PROGRAM DataTypes
VAR
	floatExample : REAL;
	someStr : STRING;
	someInt : INT := 20;
	{REFERENCE TO someInt}
	refInt : REFERENCE TO INT REF=someInt;
	
	bytesCountFloat : UINT;
	bytesCountInt : UINT;
	bytesCountStr : UINT;
	
	{U may declare negative indexes : [-5..4]}
	someArr : ARRAY[1..5] OF INT := [10, 20, 30, 40, 50];
	twoDemArr : ARRAY [0..3, 0..9] OF REAL;
END_VAR

bytesCountFloat := SIZEOF(floatExample);
bytesCountStr := SIZEOF(someStr);
bytesCountInt := SIZEOF(someInt);

someArr[2] := 0;

END_PROGRAM

(* stored: Version 1.1.0.1, ProductVersion 3.1.4024.11
   POU DataTypes: Id {aa884303-2ff6-4018-8688-1781a7e4f9d8}, SpecialFunc None *)
